{attribute addProperty BoxType "EK1100-0000-0018"}
{attribute addProperty Id "Beckhoff_EL3xxxEK1122Beckhoff_EL3xxxEK1122_9FE29313162A_0001_EL3602_0000_0016EL3602_9C69A51A27234A_0002_EL3602_0000_0017EL3602_9C69A51A27234A_0003_EL3602_0000_0018EL3602_9C69A51A27234A_0004_EL3602_0000_0019EL3602_9C69A51A27234A_0005_EL3602_0002_0016EL3602_4869176519224A_0006_EL3602_0002_0017EL3602_4869176519224A_0007_EL3602_0002_0018EL3602_4869176519224A_0008_EL3602_0010_0016EL3602_9C69A51A27234A_0009_EL3602_0010_0017EL3602_9C69A51A27234A_0010_EL3602_0010_0018EL3602_9C69A51A27234A_0011_EL3602_0010_0019EL3602_9C69A51A27234A_0012_EL3602_0020_0018EL3602_8DE8406E29036.25A_0013_EL3611_1030_0016EL3611_083DA56914418A_0014_EL3611_1030_0017EL3611_083DA56914418A_0015_EL3612_0000_0016EL3612_9C69A51A27234A_0016_EL3612_0000_0017EL3612_9C69A51A27234A_0017_EL3612_0000_0018EL3612_9C69A51A27234A_0018_EL3612_0000_0019EL3612_9C69A51A27234A_0019_EL3612_0020_0018EL3612_9C69A51A27234A_0020_EL3612_0020_0019EL3612_9C69A51A27234A_0021_EL3621_0020_0016EL3621_85E9A03514418A_0022_EL3621_0020_0017EL3621_85E9A03514418A_0023_EL3632_0000_0016EL3632_817473E359274A_0024_EL3632_0000_0017EL3632_817473E359274A_0025_EL3632_0000_0018EL3632_817473E359274A_0026_EL3632_0000_0019EL3632_817473E359274A_0027_EL3632_0000_0020EL3632_817473E359274A_0028_EL3632_0000_0021EL3632_817473E359274A_0029_EL3632_0000_0022EL3632_C340233D59274A_0030_EL3632_0000_0023EL3632_C340233D59274A_0031_EL3681_0000_0017EL3681_494E7C6C17622A_0032_EL3681_0000_0018EL3681_7DAD71F717622A_0033_EL3681_0000_0019EL3681_7DAD71F717622A_0034_EL3681_0000_0020EL3681_AEC4272017622A_0035_EL3681_0000_0021EL3681_01269A6017622A_0036_EL3692_0000_0017EL3692_E9B845C428836A_0037_EL3692_0000_0018EL3692_E9B845C428836A_0038_EL3692_0000_0019EL3692_E9B845C428836A_0039_EL3692_0000_0020EL3692_3E4349A528836A_0040_EL3692_0000_0021EL3692_3E4349A528836"}
{attribute addProperty CRC "2394328244"}
{attribute addProperty SizeInBites "12322"}
{attribute addProperty SizeInBytes "1540.25"}
TYPE Beckhoff_EL3xxx_8EB68CB4 EXTENDS EK1100_179A0949 :
STRUCT
	{attribute addProperty Name "Beckhoff_EL3xxxEK1122"}
	Beckhoff_EL3xxxEK1122 : Beckhoff_EL3xxxEK1122_9FE29313;
	{attribute addProperty Name "A_0001_EL3602_0000_0016"}
	A_0001_EL3602_0000_0016 : EL3602_9C69A51A;
	{attribute addProperty Name "A_0002_EL3602_0000_0017"}
	A_0002_EL3602_0000_0017 : EL3602_9C69A51A;
	{attribute addProperty Name "A_0003_EL3602_0000_0018"}
	A_0003_EL3602_0000_0018 : EL3602_9C69A51A;
	{attribute addProperty Name "A_0004_EL3602_0000_0019"}
	A_0004_EL3602_0000_0019 : EL3602_9C69A51A;
	{attribute addProperty Name "A_0005_EL3602_0002_0016"}
	A_0005_EL3602_0002_0016 : EL3602_48691765;
	{attribute addProperty Name "A_0006_EL3602_0002_0017"}
	A_0006_EL3602_0002_0017 : EL3602_48691765;
	{attribute addProperty Name "A_0007_EL3602_0002_0018"}
	A_0007_EL3602_0002_0018 : EL3602_48691765;
	{attribute addProperty Name "A_0008_EL3602_0010_0016"}
	A_0008_EL3602_0010_0016 : EL3602_9C69A51A;
	{attribute addProperty Name "A_0009_EL3602_0010_0017"}
	A_0009_EL3602_0010_0017 : EL3602_9C69A51A;
	{attribute addProperty Name "A_0010_EL3602_0010_0018"}
	A_0010_EL3602_0010_0018 : EL3602_9C69A51A;
	{attribute addProperty Name "A_0011_EL3602_0010_0019"}
	A_0011_EL3602_0010_0019 : EL3602_9C69A51A;
	{attribute addProperty Name "A_0012_EL3602_0020_0018"}
	A_0012_EL3602_0020_0018 : EL3602_8DE8406E;
	{attribute addProperty Name "A_0013_EL3611_1030_0016"}
	A_0013_EL3611_1030_0016 : EL3611_083DA569;
	{attribute addProperty Name "A_0014_EL3611_1030_0017"}
	A_0014_EL3611_1030_0017 : EL3611_083DA569;
	{attribute addProperty Name "A_0015_EL3612_0000_0016"}
	A_0015_EL3612_0000_0016 : EL3612_9C69A51A;
	{attribute addProperty Name "A_0016_EL3612_0000_0017"}
	A_0016_EL3612_0000_0017 : EL3612_9C69A51A;
	{attribute addProperty Name "A_0017_EL3612_0000_0018"}
	A_0017_EL3612_0000_0018 : EL3612_9C69A51A;
	{attribute addProperty Name "A_0018_EL3612_0000_0019"}
	A_0018_EL3612_0000_0019 : EL3612_9C69A51A;
	{attribute addProperty Name "A_0019_EL3612_0020_0018"}
	A_0019_EL3612_0020_0018 : EL3612_9C69A51A;
	{attribute addProperty Name "A_0020_EL3612_0020_0019"}
	A_0020_EL3612_0020_0019 : EL3612_9C69A51A;
	{attribute addProperty Name "A_0021_EL3621_0020_0016"}
	A_0021_EL3621_0020_0016 : EL3621_85E9A035;
	{attribute addProperty Name "A_0022_EL3621_0020_0017"}
	A_0022_EL3621_0020_0017 : EL3621_85E9A035;
	{attribute addProperty Name "A_0023_EL3632_0000_0016"}
	A_0023_EL3632_0000_0016 : EL3632_817473E3;
	{attribute addProperty Name "A_0024_EL3632_0000_0017"}
	A_0024_EL3632_0000_0017 : EL3632_817473E3;
	{attribute addProperty Name "A_0025_EL3632_0000_0018"}
	A_0025_EL3632_0000_0018 : EL3632_817473E3;
	{attribute addProperty Name "A_0026_EL3632_0000_0019"}
	A_0026_EL3632_0000_0019 : EL3632_817473E3;
	{attribute addProperty Name "A_0027_EL3632_0000_0020"}
	A_0027_EL3632_0000_0020 : EL3632_817473E3;
	{attribute addProperty Name "A_0028_EL3632_0000_0021"}
	A_0028_EL3632_0000_0021 : EL3632_817473E3;
	{attribute addProperty Name "A_0029_EL3632_0000_0022"}
	A_0029_EL3632_0000_0022 : EL3632_C340233D;
	{attribute addProperty Name "A_0030_EL3632_0000_0023"}
	A_0030_EL3632_0000_0023 : EL3632_C340233D;
	{attribute addProperty Name "A_0031_EL3681_0000_0017"}
	A_0031_EL3681_0000_0017 : EL3681_494E7C6C;
	{attribute addProperty Name "A_0032_EL3681_0000_0018"}
	A_0032_EL3681_0000_0018 : EL3681_7DAD71F7;
	{attribute addProperty Name "A_0033_EL3681_0000_0019"}
	A_0033_EL3681_0000_0019 : EL3681_7DAD71F7;
	{attribute addProperty Name "A_0034_EL3681_0000_0020"}
	A_0034_EL3681_0000_0020 : EL3681_AEC42720;
	{attribute addProperty Name "A_0035_EL3681_0000_0021"}
	A_0035_EL3681_0000_0021 : EL3681_01269A60;
	{attribute addProperty Name "A_0036_EL3692_0000_0017"}
	A_0036_EL3692_0000_0017 : EL3692_E9B845C4;
	{attribute addProperty Name "A_0037_EL3692_0000_0018"}
	A_0037_EL3692_0000_0018 : EL3692_E9B845C4;
	{attribute addProperty Name "A_0038_EL3692_0000_0019"}
	A_0038_EL3692_0000_0019 : EL3692_E9B845C4;
	{attribute addProperty Name "A_0039_EL3692_0000_0020"}
	A_0039_EL3692_0000_0020 : EL3692_3E4349A5;
	{attribute addProperty Name "A_0040_EL3692_0000_0021"}
	A_0040_EL3692_0000_0021 : EL3692_3E4349A5;
END_STRUCT
END_TYPE

(* stored: Version 1.2.0.0, ProductVersion 3.1.4024.9
   DUT Beckhoff_EL3xxx_8EB68CB4: Id {7d2e33e3-cc16-4f8a-b8cc-e2c0b3eaacc8} *)
